// TIA Portal project "AP2_s71200" (V14)

(* hardware
DEVICE "S7-1200 station_1"  S7-1200 Station
   slot 0: "Rack_0"  S7-1200 Rack  Rack  V1.0
   slot 1: "PLC_1"  CPU 1214C DC/DC/DC  6ES7 214-1AG40-0XB0  V4.2
   slot 2: "DI 16/DQ 16x24VDC_1"  6ES7 223-1BL32-0XB0  V2.0
*)

// ===== PLC "PLC_1"  CPU 1214C DC/DC/DC =====

VAR_GLOBAL   // PLC tag table "Default tag table"
   "-F5" AT %I0.0 : Bool;
   "-S3" AT %I0.1 : Bool;
   "-S4" AT %I0.2 : Bool;
   "-S5" AT %I0.3 : Bool;
   "-S6" AT %I0.4 : Bool;
   "-S7" AT %I0.5 : Bool;
   "-S8" AT %I0.6 : Bool;
   "-S9" AT %I0.7 : Bool;
   "-S10" AT %I1.0 : Bool;
   "-S11" AT %I1.1 : Bool;
   "-S12" AT %I1.2 : Bool;
   "-BP1" AT %I1.3 : Bool;
   "-B11" AT %I1.4 : Bool;
   "-B12" AT %I1.5 : Bool;
   "-B13" AT %I2.0 : Bool;
   "-B21" AT %I2.1 : Bool;
   "-B22" AT %I2.2 : Bool;
   "-B31" AT %I2.3 : Bool;
   "-B32" AT %I2.4 : Bool;
   "Reserve1" AT %I2.5 : Bool;
   "Reserve2" AT %I2.6 : Bool;
   "Reserve3" AT %I2.7 : Bool;
   "Reserve4" AT %I3.0 : Bool;
   "-F7" AT %I3.1 : Bool;
   "-M21" AT %Q0.0 : Bool;
   "-M22" AT %Q0.1 : Bool;
   "-M31" AT %Q0.2 : Bool;
   "-M32" AT %Q0.3 : Bool;
   "Reserve5" AT %Q0.4 : Bool;
   "Reserve6" AT %Q0.5 : Bool;
   "-Q5" AT %Q0.6 : Bool;
   "-Q6" AT %Q0.7 : Bool;
   "-P32" AT %Q2.0 : Bool;
   "Reserve7" AT %Q2.1 : Bool;
   "-Q60" AT %Q2.2 : Bool;
   "-P2" AT %Q2.3 : Bool;
   "-P3" AT %Q2.4 : Bool;
   "-P4" AT %Q2.5 : Bool;
   "-P5" AT %Q2.6 : Bool;
   "-P6" AT %Q2.7 : Bool;
   "-P7" AT %Q3.0 : Bool;
   "-P8" AT %Q3.1 : Bool;
   "-P10" AT %Q3.2 : Bool;
   "-P11" AT %Q3.3 : Bool;
   "-P12" AT %Q3.4 : Bool;
   "-P13" AT %Q3.5 : Bool;
   "-P14" AT %Q3.6 : Bool;
   "-Reserve8" AT %Q3.7 : Bool;
   "G_Notification" AT %M0.0 : Bool;
   "G_Allow" AT %M0.1 : Bool;
   "Button" AT %M0.3 : Bool;
   "Auto" AT %M0.4 : Bool;
   "Allow" AT %M0.5 : Bool;
   "1Hz" AT %M0.6 : Bool;
   "T_Block" AT %M0.7 : Bool;
   "M21_A" AT %M1.0 : Bool;
   "M22_A" AT %M1.1 : Bool;
   "M31_A" AT %M1.2 : Bool;
   "M32_A" AT %M1.3 : Bool;
   "Q5_A" AT %M1.4 : Bool;
   "Q6_A" AT %M1.5 : Bool;
   "Q60_A" AT %M1.6 : Bool;
   "M21_B" AT %M1.7 : Bool;
   "M22_B" AT %M2.0 : Bool;
   "M31_B" AT %M2.1 : Bool;
   "M32_B" AT %M2.2 : Bool;
   "Q5_B" AT %M2.3 : Bool;
   "Q6_B" AT %M2.4 : Bool;
   "Q60_B" AT %M2.5 : Bool;
   "Out_Step 3" AT %M0.2 : Bool;
END_VAR

DATA_BLOCK "Clock_DB"   // DB3
{ S7_Optimized_Access := 'TRUE' }
VERSION : 0.1
// stored: InstanceOfName Clock
"Clock"
BEGIN
END_DATA_BLOCK

DATA_BLOCK "Safety_Activation_DB"   // DB4
{ S7_Optimized_Access := 'TRUE' }
VERSION : 0.1
// stored: InstanceOfName Safety_Activation
"Safety_Activation"
BEGIN
END_DATA_BLOCK

DATA_BLOCK "G_Allow__DB"   // DB5
{ S7_Optimized_Access := 'TRUE' }
VERSION : 0.1
// stored: InstanceOfName G_Allow_
"G_Allow_"
BEGIN
END_DATA_BLOCK

DATA_BLOCK "G_T_Block_DB"   // DB6
{ S7_Optimized_Access := 'TRUE' }
VERSION : 0.1
// stored: InstanceOfName G_T_Block
"G_T_Block"
BEGIN
END_DATA_BLOCK

DATA_BLOCK "G_Button_DB"   // DB7
{ S7_Optimized_Access := 'TRUE' }
VERSION : 0.1
// stored: InstanceOfName G_Button
"G_Button"
BEGIN
END_DATA_BLOCK

DATA_BLOCK "G_Notifications_DB"   // DB8
{ S7_Optimized_Access := 'TRUE' }
VERSION : 0.1
// stored: InstanceOfName G_Notifications
"G_Notifications"
BEGIN
END_DATA_BLOCK

DATA_BLOCK "G_Auto_DB"   // DB21
{ S7_Optimized_Access := 'TRUE' }
VERSION : 0.1
// stored: InstanceOfName G_Auto
"G_Auto"
BEGIN
END_DATA_BLOCK

DATA_BLOCK "Output_DB"   // DB22
{ S7_Optimized_Access := 'TRUE' }
VERSION : 0.1
// stored: InstanceOfName Output
"Output"
BEGIN
END_DATA_BLOCK

// folder: System blocks/Program resources

DATA_BLOCK "0.5s/X500"   // DB1
{ S7_Optimized_Access := 'TRUE' }
AUTHOR : Simatic
FAMILY : IEC
NAME : IEC_TMR
VERSION : 1.0
// stored: InstanceOfName IEC_TIMER
"IEC_TIMER"
BEGIN
END_DATA_BLOCK

DATA_BLOCK "0.5s/X501"   // DB2
{ S7_Optimized_Access := 'TRUE' }
AUTHOR : Simatic
FAMILY : IEC
NAME : IEC_TMR
VERSION : 1.0
// stored: InstanceOfName IEC_TIMER
"IEC_TIMER"
BEGIN
END_DATA_BLOCK

DATA_BLOCK "1s/B11_X301"   // DB9
{ S7_Optimized_Access := 'TRUE' }
AUTHOR : Simatic
FAMILY : IEC
NAME : IEC_TMR
VERSION : 1.0
// stored: InstanceOfName IEC_TIMER
"IEC_TIMER"
BEGIN
END_DATA_BLOCK

DATA_BLOCK "2s/B22_X302"   // DB10
{ S7_Optimized_Access := 'TRUE' }
AUTHOR : Simatic
FAMILY : IEC
NAME : IEC_TMR
VERSION : 1.0
// stored: InstanceOfName IEC_TIMER
"IEC_TIMER"
BEGIN
END_DATA_BLOCK

DATA_BLOCK "1s/B21_X303"   // DB11
{ S7_Optimized_Access := 'TRUE' }
AUTHOR : Simatic
FAMILY : IEC
NAME : IEC_TMR
VERSION : 1.0
// stored: InstanceOfName IEC_TIMER
"IEC_TIMER"
BEGIN
END_DATA_BLOCK

DATA_BLOCK "1s/B12_X304"   // DB12
{ S7_Optimized_Access := 'TRUE' }
AUTHOR : Simatic
FAMILY : IEC
NAME : IEC_TMR
VERSION : 1.0
// stored: InstanceOfName IEC_TIMER
"IEC_TIMER"
BEGIN
END_DATA_BLOCK

DATA_BLOCK "1s/B22_X305"   // DB13
{ S7_Optimized_Access := 'TRUE' }
AUTHOR : Simatic
FAMILY : IEC
NAME : IEC_TMR
VERSION : 1.0
// stored: InstanceOfName IEC_TIMER
"IEC_TIMER"
BEGIN
END_DATA_BLOCK

DATA_BLOCK "1s/B21_X308"   // DB14
{ S7_Optimized_Access := 'TRUE' }
AUTHOR : Simatic
FAMILY : IEC
NAME : IEC_TMR
VERSION : 1.0
// stored: InstanceOfName IEC_TIMER
"IEC_TIMER"
BEGIN
END_DATA_BLOCK

DATA_BLOCK "1s/B13_X309"   // DB15
{ S7_Optimized_Access := 'TRUE' }
AUTHOR : Simatic
FAMILY : IEC
NAME : IEC_TMR
VERSION : 1.0
// stored: InstanceOfName IEC_TIMER
"IEC_TIMER"
BEGIN
END_DATA_BLOCK

DATA_BLOCK "1s/B22_X310"   // DB16
{ S7_Optimized_Access := 'TRUE' }
AUTHOR : Simatic
FAMILY : IEC
NAME : IEC_TMR
VERSION : 1.0
// stored: InstanceOfName IEC_TIMER
"IEC_TIMER"
BEGIN
END_DATA_BLOCK

DATA_BLOCK "1s/X311"   // DB17
{ S7_Optimized_Access := 'TRUE' }
AUTHOR : Simatic
FAMILY : IEC
NAME : IEC_TMR
VERSION : 1.0
// stored: InstanceOfName IEC_TIMER
"IEC_TIMER"
BEGIN
END_DATA_BLOCK

DATA_BLOCK "1s/B21_X312"   // DB18
{ S7_Optimized_Access := 'TRUE' }
AUTHOR : Simatic
FAMILY : IEC
NAME : IEC_TMR
VERSION : 1.0
// stored: InstanceOfName IEC_TIMER
"IEC_TIMER"
BEGIN
END_DATA_BLOCK

DATA_BLOCK "2s/B31_X313"   // DB19
{ S7_Optimized_Access := 'TRUE' }
AUTHOR : Simatic
FAMILY : IEC
NAME : IEC_TMR
VERSION : 1.0
// stored: InstanceOfName IEC_TIMER
"IEC_TIMER"
BEGIN
END_DATA_BLOCK

DATA_BLOCK "1s/B32_X314"   // DB20
{ S7_Optimized_Access := 'TRUE' }
AUTHOR : Simatic
FAMILY : IEC
NAME : IEC_TMR
VERSION : 1.0
// stored: InstanceOfName IEC_TIMER
"IEC_TIMER"
BEGIN
END_DATA_BLOCK

// folder: (top level)

FUNCTION_BLOCK "Safety_Activation"   // FB1, FBD
{ S7_Optimized_Access := 'TRUE' }
VERSION : 0.1
   VAR_INPUT
      Allow : Bool;
      BP1 : Bool;
      S3 : Bool;
      S4 : Bool;
      F5 : Bool;
      F7 : Bool;
   END_VAR
   VAR_OUTPUT
      G_Notifications : Bool;
      G_Allow : Bool;
      "Out_step 3" : Bool;
      Button : Bool;
      Auto : Bool;
   END_VAR
   VAR
      "Step 1" : Bool;
      "Step 2" : Bool;
      "Step 3" : Bool;
      "Step 4" : Bool;
      "Step 5" : Bool;
   END_VAR
BEGIN

REGION Network 1
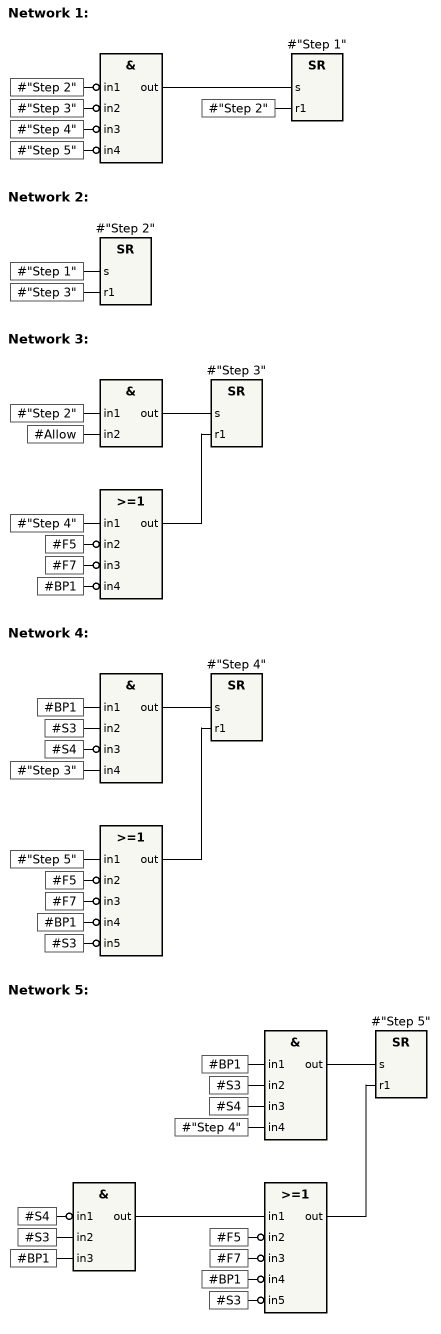
   IF NOT #"Step 2" AND NOT #"Step 3" AND NOT #"Step 4" AND NOT #"Step 5" THEN
       #"Step 1" := TRUE;   // SR flip-flop
   END_IF;
   IF #"Step 2" THEN #"Step 1" := FALSE; END_IF;
END_REGION

REGION Network 2
   IF #"Step 1" THEN
       #"Step 2" := TRUE;   // SR flip-flop
   END_IF;
   IF #"Step 3" THEN #"Step 2" := FALSE; END_IF;
END_REGION

REGION Network 3
   IF #"Step 2" AND #Allow THEN
       #"Step 3" := TRUE;   // SR flip-flop
   END_IF;
   IF #"Step 4" OR NOT #F5 OR NOT #F7 OR NOT #BP1 THEN #"Step 3" := FALSE; END_IF;
END_REGION

REGION Network 4
   IF #BP1 AND #S3 AND NOT #S4 AND #"Step 3" THEN
       #"Step 4" := TRUE;   // SR flip-flop
   END_IF;
   IF #"Step 5" OR NOT #F5 OR NOT #F7 OR NOT #BP1 OR NOT #S3 THEN #"Step 4" := FALSE; END_IF;
END_REGION

REGION Network 5
   IF #BP1 AND #S3 AND #S4 AND #"Step 4" THEN
       #"Step 5" := TRUE;   // SR flip-flop
   END_IF;
   IF (NOT #S4 AND #S3 AND #BP1) OR NOT #F5 OR NOT #F7 OR NOT #BP1 OR NOT #S3 THEN
       #"Step 5" := FALSE;
   END_IF;
END_REGION

REGION Network 6
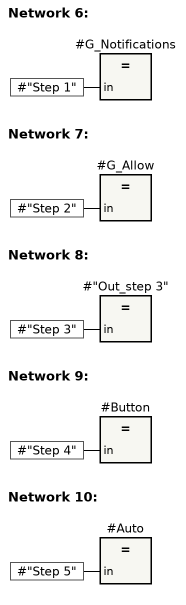
   #G_Notifications := #"Step 1";
END_REGION

REGION Network 7
   #G_Allow := #"Step 2";
END_REGION

REGION Network 8
   #"Out_step 3" := #"Step 3";
END_REGION

REGION Network 9
   #Button := #"Step 4";
END_REGION

REGION Network 10
   #Auto := #"Step 5";
END_REGION
END_FUNCTION_BLOCK

FUNCTION_BLOCK "Clock"   // FB2, FBD
{ S7_Optimized_Access := 'TRUE' }
VERSION : 0.1
   VAR_OUTPUT
      "1Hz" : Bool;
   END_VAR
   VAR
      "Step 500" : Bool;
      "Step 501" : Bool;
   END_VAR
BEGIN

REGION Network 1
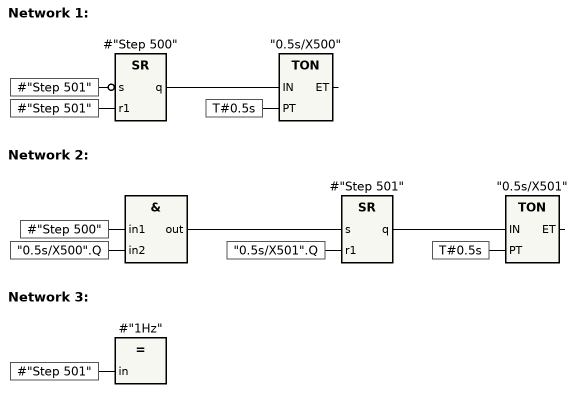
   IF NOT #"Step 501" THEN
       #"Step 500" := TRUE;   // SR flip-flop
   END_IF;
   IF #"Step 501" THEN #"Step 500" := FALSE; END_IF;
   "0.5s/X500".TON(IN := #"Step 500", PT := T#0.5s);
END_REGION

REGION Network 2
   IF #"Step 500" AND "0.5s/X500".Q THEN
       #"Step 501" := TRUE;   // SR flip-flop
   END_IF;
   IF "0.5s/X501".Q THEN #"Step 501" := FALSE; END_IF;
   "0.5s/X501".TON(IN := #"Step 501", PT := T#0.5s);
END_REGION

REGION Network 3
   #"1Hz" := #"Step 501";
END_REGION
END_FUNCTION_BLOCK

FUNCTION_BLOCK "G_Allow_"   // FB3, FBD
{ S7_Optimized_Access := 'TRUE' }
VERSION : 0.1
   VAR_INPUT
      G_Allow : Bool;
      "Out_step 3" : Bool;
      F5 : Bool;
      F7 : Bool;
      S4 : Bool;
      S5 : Bool;
      S6 : Bool;
      S7 : Bool;
      S8 : Bool;
      S9 : Bool;
      S10 : Bool;
      S12 : Bool;
   END_VAR
   VAR_OUTPUT
      Allow : Bool;
   END_VAR
   VAR
      "Step 50" : Bool;
      "Step 51" : Bool;
   END_VAR
BEGIN

REGION Network 1
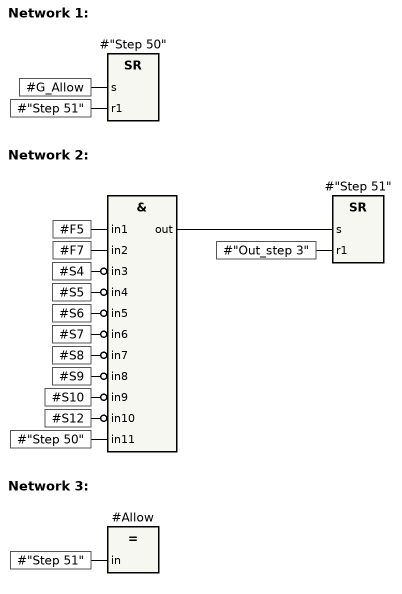
   IF #G_Allow THEN
       #"Step 50" := TRUE;   // SR flip-flop
   END_IF;
   IF #"Step 51" THEN #"Step 50" := FALSE; END_IF;
END_REGION

REGION Network 2
   IF #F5 AND #F7 AND NOT #S4 AND NOT #S5 AND NOT #S6 AND NOT #S7 AND NOT #S8 AND NOT #S9 AND NOT #S10 AND NOT #S12 AND #"Step 50" THEN
       #"Step 51" := TRUE;   // SR flip-flop
   END_IF;
   IF #"Out_step 3" THEN #"Step 51" := FALSE; END_IF;
END_REGION

REGION Network 3
   #Allow := #"Step 51";
END_REGION
END_FUNCTION_BLOCK

FUNCTION_BLOCK "G_T_Block"   // FB4, FBD
{ S7_Optimized_Access := 'TRUE' }
VERSION : 0.1
   VAR_INPUT
      Button : Bool;
      S6 : Bool;
      S7 : Bool;
   END_VAR
   VAR_OUTPUT
      T_Block : Bool;
   END_VAR
   VAR
      "Step 400" : Bool;
      "Step 401" : Bool;
   END_VAR
BEGIN

REGION Network 1
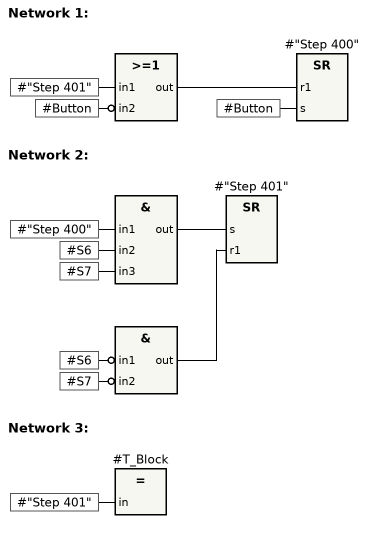
   IF #Button THEN
       #"Step 400" := TRUE;   // SR flip-flop
   END_IF;
   IF #"Step 401" OR NOT #Button THEN #"Step 400" := FALSE; END_IF;
END_REGION

REGION Network 2
   IF #"Step 400" AND #S6 AND #S7 THEN
       #"Step 401" := TRUE;   // SR flip-flop
   END_IF;
   IF NOT #S6 AND NOT #S7 THEN #"Step 401" := FALSE; END_IF;
END_REGION

REGION Network 3
   #T_Block := #"Step 401";
END_REGION
END_FUNCTION_BLOCK

FUNCTION_BLOCK "G_Button"   // FB5, FBD
{ S7_Optimized_Access := 'TRUE' }
VERSION : 0.1
   VAR_INPUT
      G_Button : Bool;
      G_T_Block : Bool;
      S6 : Bool;
      S7 : Bool;
      S8 : Bool;
      S9 : Bool;
      S10 : Bool;
      S12 : Bool;
      B11 : Bool;
      B13 : Bool;
      B21 : Bool;
      B22 : Bool;
      B31 : Bool;
      B32 : Bool;
      "Q5.in" : Bool;
      "Q6.in" : Bool;
   END_VAR
   VAR_OUTPUT
      Q5_B : Bool;
      Q6_B : Bool;
      M21_B : Bool;
      M22_B : Bool;
      M31_B : Bool;
      M32_B : Bool;
      Q60_B : Bool;
   END_VAR
   VAR
      "Step 200" : Bool;
   END_VAR
BEGIN

REGION Network 1
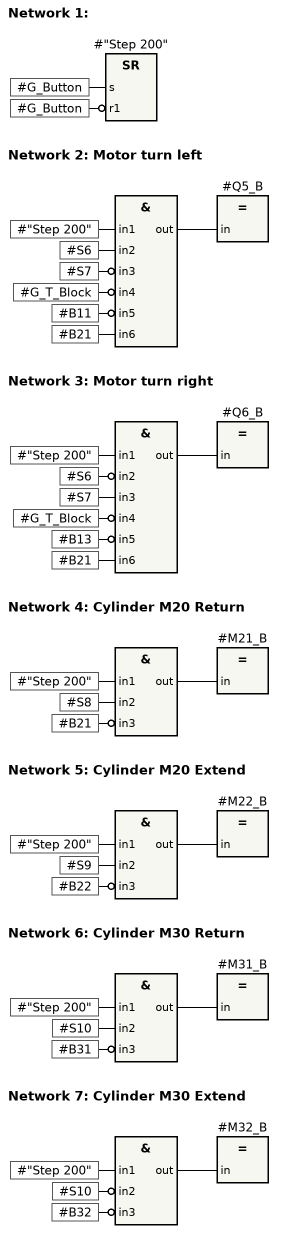
   IF #G_Button THEN
       #"Step 200" := TRUE;   // SR flip-flop
   END_IF;
   IF NOT #G_Button THEN #"Step 200" := FALSE; END_IF;
END_REGION

REGION Network 2: Motor turn left
   #Q5_B := #"Step 200" AND #S6 AND NOT #S7 AND NOT #G_T_Block AND NOT #B11 AND #B21;
END_REGION

REGION Network 3: Motor turn right
   #Q6_B := #"Step 200" AND NOT #S6 AND #S7 AND NOT #G_T_Block AND NOT #B13 AND #B21;
END_REGION

REGION Network 4: Cylinder M20 Return
   #M21_B := #"Step 200" AND #S8 AND NOT #B21;
END_REGION

REGION Network 5: Cylinder M20 Extend
   #M22_B := #"Step 200" AND #S9 AND NOT #B22;
END_REGION

REGION Network 6: Cylinder M30 Return
   #M31_B := #"Step 200" AND #S10 AND NOT #B31;
END_REGION

REGION Network 7: Cylinder M30 Extend
   #M32_B := #"Step 200" AND NOT #S10 AND NOT #B32;
END_REGION

REGION Network 8: Demagnetization
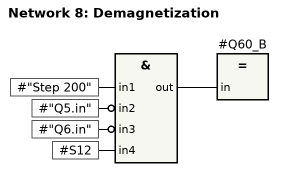
   #Q60_B := #"Step 200" AND NOT #"Q5.in" AND NOT #"Q6.in" AND #S12;
END_REGION
END_FUNCTION_BLOCK

FUNCTION_BLOCK "G_Notifications"   // FB6, FBD
{ S7_Optimized_Access := 'TRUE' }
VERSION : 0.1
   VAR_INPUT
      S3 : Bool;
      G_Notification : Bool;
      Auto : Bool;
      Button : Bool;
      "1Hz" : Bool;
      F7 : Bool;
      BP1 : Bool;
      B11 : Bool;
      B12 : Bool;
      B13 : Bool;
      B21 : Bool;
      B22 : Bool;
      B31 : Bool;
      B32 : Bool;
      "Q5.in" : Bool;
      "Q6.in" : Bool;
      "Q60.in" : Bool;
   END_VAR
   VAR_OUTPUT
      P2 : Bool;
      P3 : Bool;
      P4 : Bool;
      P5 : Bool;
      P6 : Bool;
      P7 : Bool;
      P8 : Bool;
      P10 : Bool;
      P11 : Bool;
      P12 : Bool;
      P13 : Bool;
      P14 : Bool;
      P32 : Bool;
   END_VAR
   VAR
      "Step 100" : Bool;
      "Step 101" : Bool;
   END_VAR
BEGIN

REGION Network 1
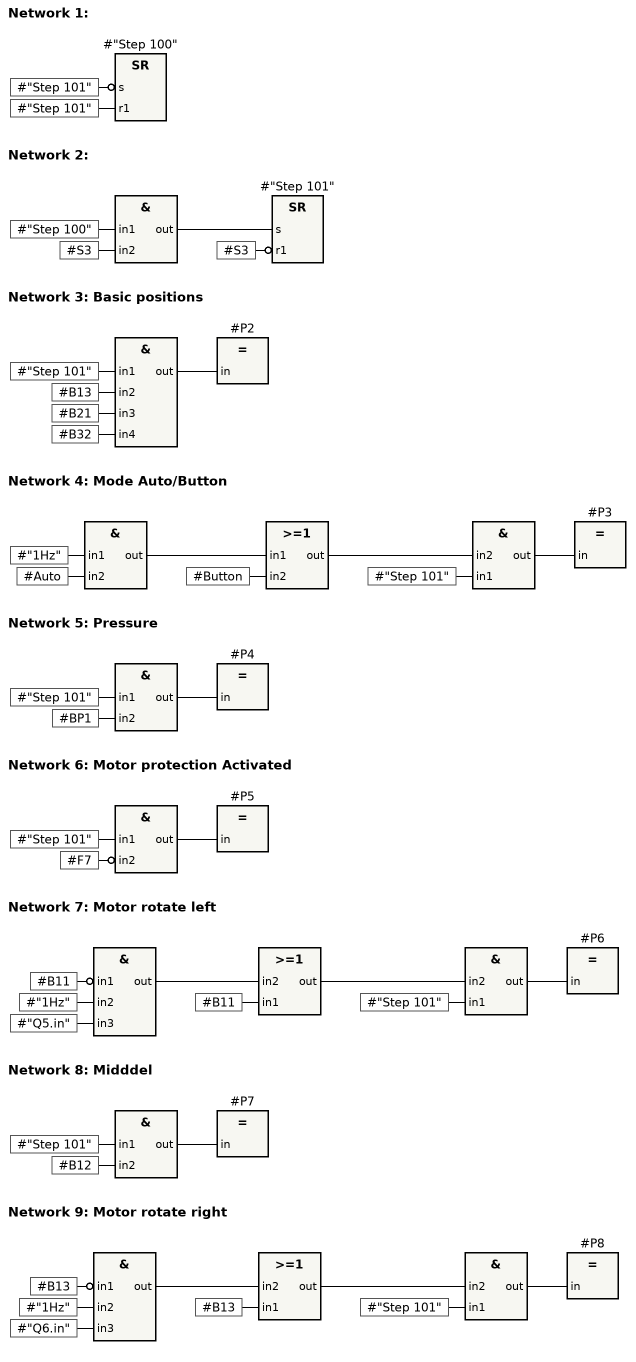
   IF NOT #"Step 101" THEN
       #"Step 100" := TRUE;   // SR flip-flop
   END_IF;
   IF #"Step 101" THEN #"Step 100" := FALSE; END_IF;
END_REGION

REGION Network 2
   IF #"Step 100" AND #S3 THEN
       #"Step 101" := TRUE;   // SR flip-flop
   END_IF;
   IF NOT #S3 THEN #"Step 101" := FALSE; END_IF;
END_REGION

REGION Network 3: Basic positions
   #P2 := #"Step 101" AND #B13 AND #B21 AND #B32;
END_REGION

REGION Network 4: Mode Auto/Button
   #P3 := ((#"1Hz" AND #Auto) OR #Button) AND #"Step 101";
END_REGION

REGION Network 5: Pressure
   #P4 := #"Step 101" AND #BP1;
END_REGION

REGION Network 6: Motor protection Activated
   #P5 := #"Step 101" AND NOT #F7;
END_REGION

REGION Network 7: Motor rotate left
   #P6 := ((NOT #B11 AND #"1Hz" AND #"Q5.in") OR #B11) AND #"Step 101";
END_REGION

REGION Network 8: Midddel
   #P7 := #"Step 101" AND #B12;
END_REGION

REGION Network 9: Motor rotate right
   #P8 := ((NOT #B13 AND #"1Hz" AND #"Q6.in") OR #B13) AND #"Step 101";
END_REGION

REGION Network 10: M20 In
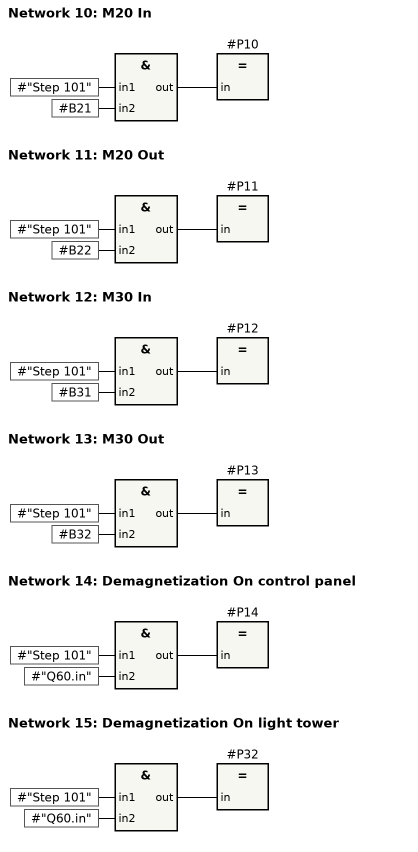
   #P10 := #"Step 101" AND #B21;
END_REGION

REGION Network 11: M20 Out
   #P11 := #"Step 101" AND #B22;
END_REGION

REGION Network 12: M30 In
   #P12 := #"Step 101" AND #B31;
END_REGION

REGION Network 13: M30 Out
   // ADD In
   #P13 := #"Step 101" AND #B32;
END_REGION

REGION Network 14: Demagnetization On control panel
   #P14 := #"Step 101" AND #"Q60.in";
END_REGION

REGION Network 15: Demagnetization On light tower
   #P32 := #"Step 101" AND #"Q60.in";
END_REGION
END_FUNCTION_BLOCK

FUNCTION_BLOCK "G_Auto"   // FB7, FBD
{ S7_Optimized_Access := 'TRUE' }
VERSION : 0.1
   VAR_INPUT
      Auto : Bool;
      S5 : Bool;
      B11 : Bool;
      B12 : Bool;
      B13 : Bool;
      B21 : Bool;
      B22 : Bool;
      B31 : Bool;
      B32 : Bool;
   END_VAR
   VAR_OUTPUT
      M21_A : Bool;
      M22_A : Bool;
      M31_A : Bool;
      M32_A : Bool;
      Q5_A : Bool;
      Q6_A : Bool;
      Q60_A : Bool;
   END_VAR
   VAR
      "Step 300" : Bool;
      "Step 301" : Bool;
      "Step 302" : Bool;
      "Step 303" : Bool;
      "Step 304" : Bool;
      "Step 305" : Bool;
      "Step 306" : Bool;
      "Step 307" : Bool;
      "Step 308" : Bool;
      "Step 309" : Bool;
      "Step 310" : Bool;
      "Step 311" : Bool;
      "Step 312" : Bool;
      "Step 313" : Bool;
      "Step 314" : Bool;
   END_VAR
BEGIN

REGION Network 1
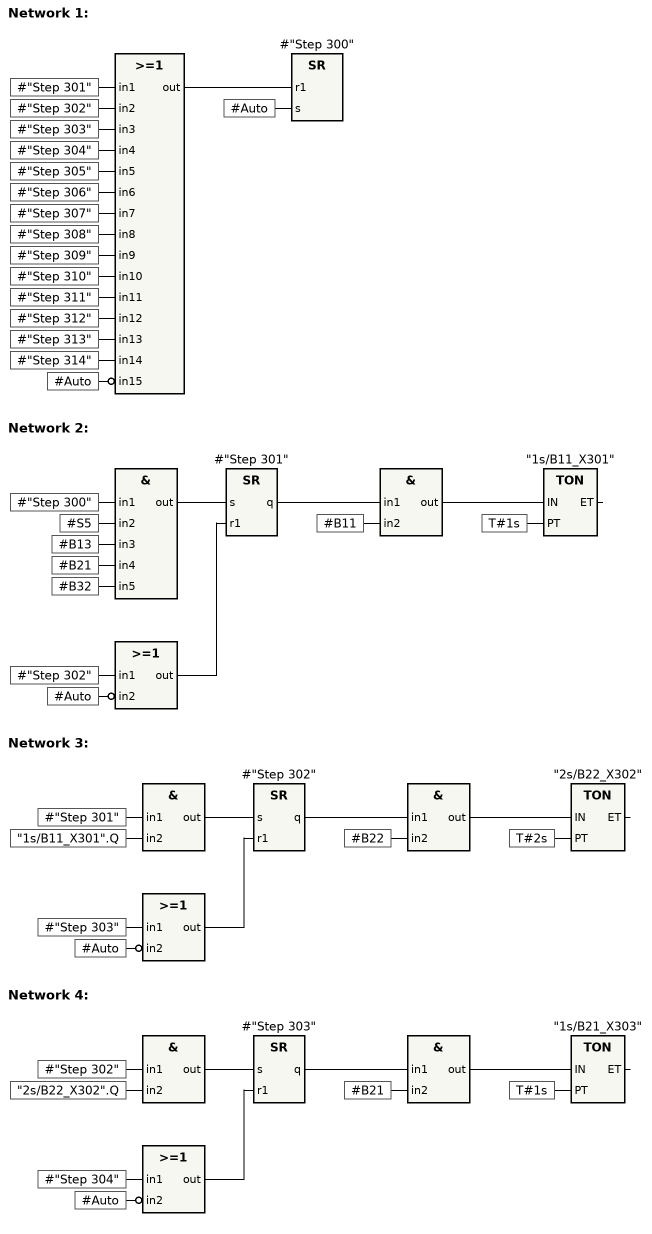
   IF #Auto THEN
       #"Step 300" := TRUE;   // SR flip-flop
   END_IF;
   IF #"Step 301" OR #"Step 302" OR #"Step 303" OR #"Step 304" OR #"Step 305" OR #"Step 306" OR #"Step 307" OR #"Step 308" OR #"Step 309" OR #"Step 310" OR #"Step 311" OR #"Step 312" OR #"Step 313" OR #"Step 314" OR NOT #Auto THEN
       #"Step 300" := FALSE;
   END_IF;
END_REGION

REGION Network 2
   IF #"Step 300" AND #S5 AND #B13 AND #B21 AND #B32 THEN
       #"Step 301" := TRUE;   // SR flip-flop
   END_IF;
   IF #"Step 302" OR NOT #Auto THEN #"Step 301" := FALSE; END_IF;
   "1s/B11_X301".TON(IN := #"Step 301" AND #B11, PT := T#1s);
END_REGION

REGION Network 3
   IF #"Step 301" AND "1s/B11_X301".Q THEN
       #"Step 302" := TRUE;   // SR flip-flop
   END_IF;
   IF #"Step 303" OR NOT #Auto THEN #"Step 302" := FALSE; END_IF;
   "2s/B22_X302".TON(IN := #"Step 302" AND #B22, PT := T#2s);
END_REGION

REGION Network 4
   IF #"Step 302" AND "2s/B22_X302".Q THEN
       #"Step 303" := TRUE;   // SR flip-flop
   END_IF;
   IF #"Step 304" OR NOT #Auto THEN #"Step 303" := FALSE; END_IF;
   "1s/B21_X303".TON(IN := #"Step 303" AND #B21, PT := T#1s);
END_REGION

REGION Network 5
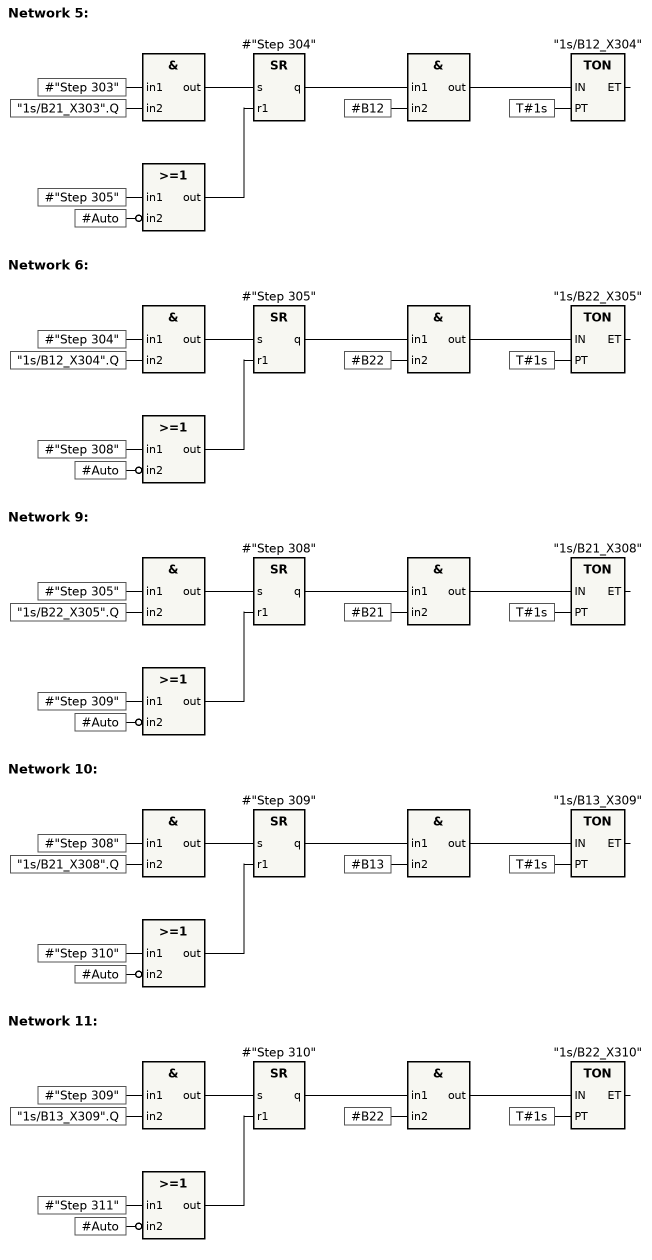
   IF #"Step 303" AND "1s/B21_X303".Q THEN
       #"Step 304" := TRUE;   // SR flip-flop
   END_IF;
   IF #"Step 305" OR NOT #Auto THEN #"Step 304" := FALSE; END_IF;
   "1s/B12_X304".TON(IN := #"Step 304" AND #B12, PT := T#1s);
END_REGION

REGION Network 6
   IF #"Step 304" AND "1s/B12_X304".Q THEN
       #"Step 305" := TRUE;   // SR flip-flop
   END_IF;
   IF #"Step 308" OR NOT #Auto THEN #"Step 305" := FALSE; END_IF;
   "1s/B22_X305".TON(IN := #"Step 305" AND #B22, PT := T#1s);
END_REGION

REGION Network 9
   IF #"Step 305" AND "1s/B22_X305".Q THEN
       #"Step 308" := TRUE;   // SR flip-flop
   END_IF;
   IF #"Step 309" OR NOT #Auto THEN #"Step 308" := FALSE; END_IF;
   "1s/B21_X308".TON(IN := #"Step 308" AND #B21, PT := T#1s);
END_REGION

REGION Network 10
   IF #"Step 308" AND "1s/B21_X308".Q THEN
       #"Step 309" := TRUE;   // SR flip-flop
   END_IF;
   IF #"Step 310" OR NOT #Auto THEN #"Step 309" := FALSE; END_IF;
   "1s/B13_X309".TON(IN := #"Step 309" AND #B13, PT := T#1s);
END_REGION

REGION Network 11
   IF #"Step 309" AND "1s/B13_X309".Q THEN
       #"Step 310" := TRUE;   // SR flip-flop
   END_IF;
   IF #"Step 311" OR NOT #Auto THEN #"Step 310" := FALSE; END_IF;
   "1s/B22_X310".TON(IN := #"Step 310" AND #B22, PT := T#1s);
END_REGION

REGION Network 12
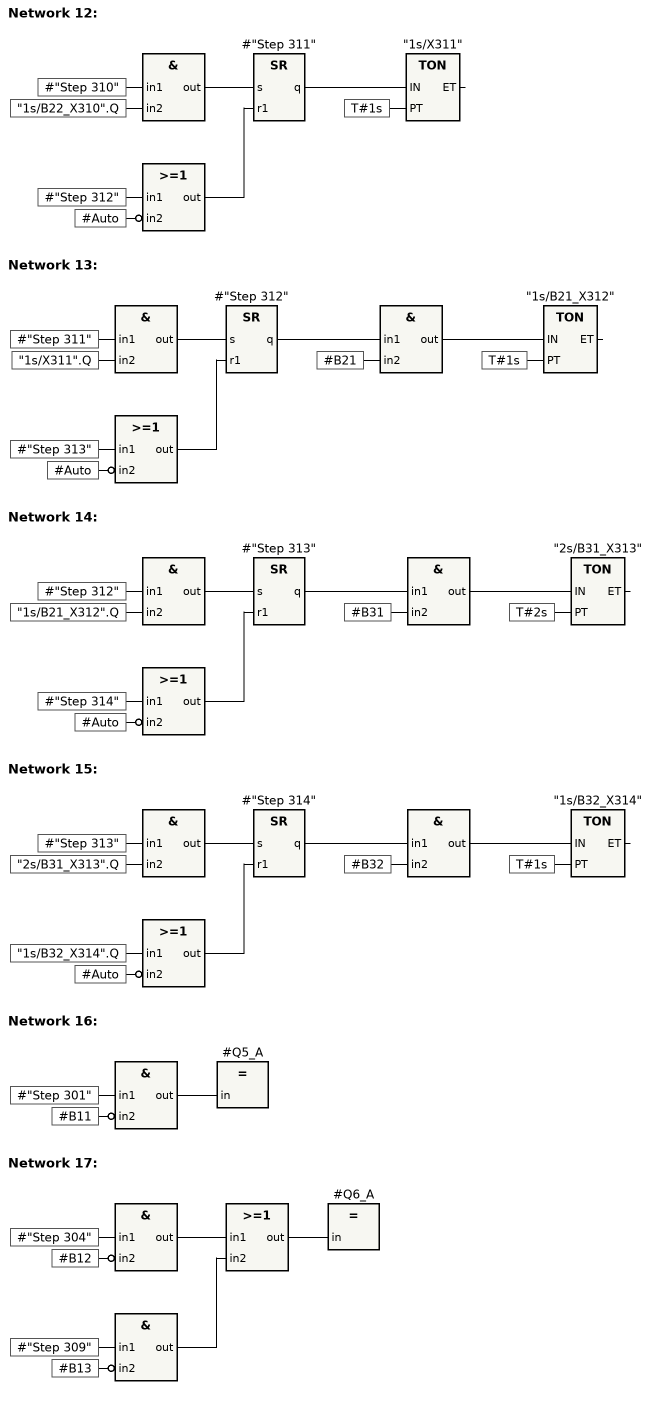
   IF #"Step 310" AND "1s/B22_X310".Q THEN
       #"Step 311" := TRUE;   // SR flip-flop
   END_IF;
   IF #"Step 312" OR NOT #Auto THEN #"Step 311" := FALSE; END_IF;
   "1s/X311".TON(IN := #"Step 311", PT := T#1s);
END_REGION

REGION Network 13
   IF #"Step 311" AND "1s/X311".Q THEN
       #"Step 312" := TRUE;   // SR flip-flop
   END_IF;
   IF #"Step 313" OR NOT #Auto THEN #"Step 312" := FALSE; END_IF;
   "1s/B21_X312".TON(IN := #"Step 312" AND #B21, PT := T#1s);
END_REGION

REGION Network 14
   IF #"Step 312" AND "1s/B21_X312".Q THEN
       #"Step 313" := TRUE;   // SR flip-flop
   END_IF;
   IF #"Step 314" OR NOT #Auto THEN #"Step 313" := FALSE; END_IF;
   "2s/B31_X313".TON(IN := #"Step 313" AND #B31, PT := T#2s);
END_REGION

REGION Network 15
   IF #"Step 313" AND "2s/B31_X313".Q THEN
       #"Step 314" := TRUE;   // SR flip-flop
   END_IF;
   IF "1s/B32_X314".Q OR NOT #Auto THEN #"Step 314" := FALSE; END_IF;
   "1s/B32_X314".TON(IN := #"Step 314" AND #B32, PT := T#1s);
END_REGION

REGION Network 16
   #Q5_A := #"Step 301" AND NOT #B11;
END_REGION

REGION Network 17
   #Q6_A := (#"Step 304" AND NOT #B12) OR (#"Step 309" AND NOT #B13);
END_REGION

REGION Network 18
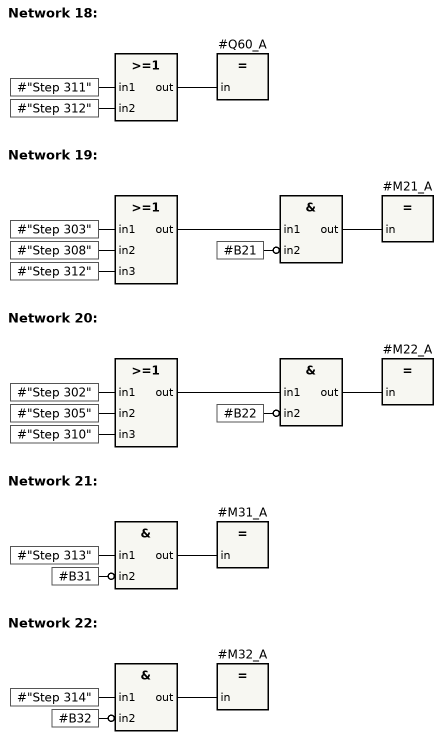
   #Q60_A := #"Step 311" OR #"Step 312";
END_REGION

REGION Network 19
   #M21_A := (#"Step 303" OR #"Step 308" OR #"Step 312") AND NOT #B21;
END_REGION

REGION Network 20
   #M22_A := (#"Step 302" OR #"Step 305" OR #"Step 310") AND NOT #B22;
END_REGION

REGION Network 21
   #M31_A := #"Step 313" AND NOT #B31;
END_REGION

REGION Network 22
   #M32_A := #"Step 314" AND NOT #B32;
END_REGION
END_FUNCTION_BLOCK

FUNCTION_BLOCK "Output"   // FB8, FBD
{ S7_Optimized_Access := 'TRUE' }
VERSION : 0.1
   VAR_INPUT
      M21_A : Bool;
      M22_A : Bool;
      M31_A : Bool;
      M32_A : Bool;
      Q5_A : Bool;
      Q6_A : Bool;
      Q60_A : Bool;
      Q5_B : Bool;
      Q6_B : Bool;
      M21_B : Bool;
      M22_B : Bool;
      M31_B : Bool;
      M32_B : Bool;
      Q60_B : Bool;
   END_VAR
   VAR_OUTPUT
      M21 : Bool;
      M22 : Bool;
      M31 : Bool;
      M32 : Bool;
      Q5 : Bool;
      Q6 : Bool;
      Q60 : Bool;
   END_VAR
BEGIN

REGION Network 1
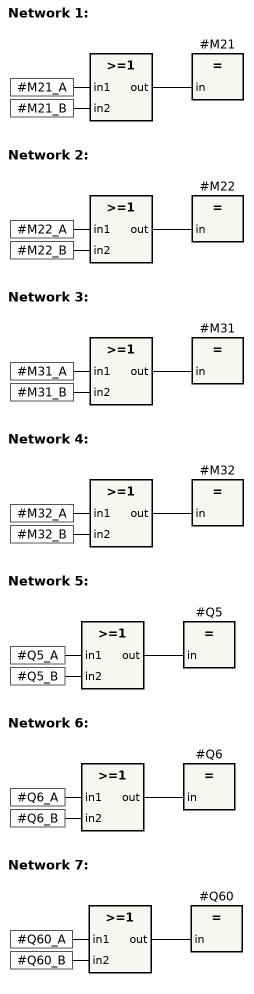
   #M21 := #M21_A OR #M21_B;
END_REGION

REGION Network 2
   #M22 := #M22_A OR #M22_B;
END_REGION

REGION Network 3
   #M31 := #M31_A OR #M31_B;
END_REGION

REGION Network 4
   #M32 := #M32_A OR #M32_B;
END_REGION

REGION Network 5
   #Q5 := #Q5_A OR #Q5_B;
END_REGION

REGION Network 6
   #Q6 := #Q6_A OR #Q6_B;
END_REGION

REGION Network 7
   #Q60 := #Q60_A OR #Q60_B;
END_REGION
END_FUNCTION_BLOCK

ORGANIZATION_BLOCK "Main"   // OB1, FBD, ProgramCycle
TITLE = "Main Program Sweep (Cycle)"
{ S7_Optimized_Access := 'TRUE' }
VERSION : 0.1
   VAR_INPUT
      Initial_Call : Bool;   // Initial call of this OB
      Remanence : Bool;   // =True, if remanent data are available
   END_VAR
BEGIN

REGION Network 1: Pluse
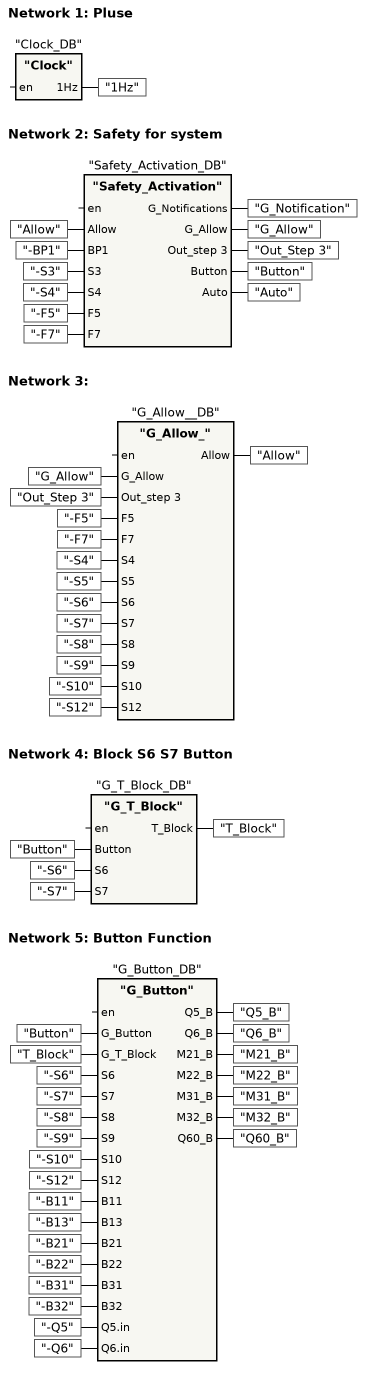
   "Clock_DB"("1Hz" => "1Hz");   // "Clock"
END_REGION

REGION Network 2: Safety for system
   "Safety_Activation_DB"(Allow := "Allow",   // "Safety_Activation"
                          BP1 := "-BP1",
                          S3 := "-S3",
                          S4 := "-S4",
                          F5 := "-F5",
                          F7 := "-F7",
                          G_Notifications => "G_Notification",
                          G_Allow => "G_Allow",
                          "Out_step 3" => "Out_Step 3",
                          Button => "Button",
                          Auto => "Auto");
END_REGION

REGION Network 3
   "G_Allow__DB"(G_Allow := "G_Allow",   // "G_Allow_"
                 "Out_step 3" := "Out_Step 3",
                 F5 := "-F5",
                 F7 := "-F7",
                 S4 := "-S4",
                 S5 := "-S5",
                 S6 := "-S6",
                 S7 := "-S7",
                 S8 := "-S8",
                 S9 := "-S9",
                 S10 := "-S10",
                 S12 := "-S12",
                 Allow => "Allow");
END_REGION

REGION Network 4: Block S6 S7 Button
   "G_T_Block_DB"(Button := "Button", S6 := "-S6", S7 := "-S7", T_Block => "T_Block");   // "G_T_Block"
END_REGION

REGION Network 5: Button Function
   "G_Button_DB"(G_Button := "Button",   // "G_Button"
                 G_T_Block := "T_Block",
                 S6 := "-S6",
                 S7 := "-S7",
                 S8 := "-S8",
                 S9 := "-S9",
                 S10 := "-S10",
                 S12 := "-S12",
                 B11 := "-B11",
                 B13 := "-B13",
                 B21 := "-B21",
                 B22 := "-B22",
                 B31 := "-B31",
                 B32 := "-B32",
                 "Q5.in" := "-Q5",
                 "Q6.in" := "-Q6",
                 Q5_B => "Q5_B",
                 Q6_B => "Q6_B",
                 M21_B => "M21_B",
                 M22_B => "M22_B",
                 M31_B => "M31_B",
                 M32_B => "M32_B",
                 Q60_B => "Q60_B");
END_REGION

REGION Network 6: Indicator
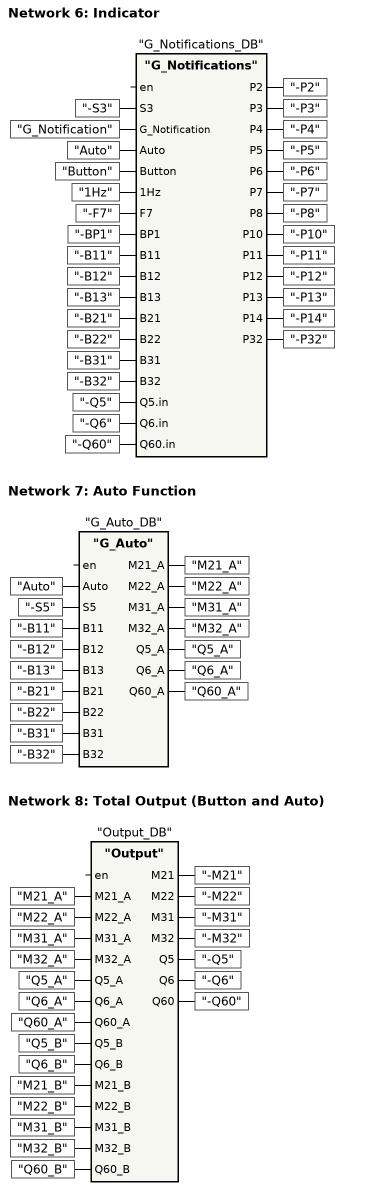
   "G_Notifications_DB"(S3 := "-S3",   // "G_Notifications"
                        G_Notification := "G_Notification",
                        Auto := "Auto",
                        Button := "Button",
                        "1Hz" := "1Hz",
                        F7 := "-F7",
                        BP1 := "-BP1",
                        B11 := "-B11",
                        B12 := "-B12",
                        B13 := "-B13",
                        B21 := "-B21",
                        B22 := "-B22",
                        B31 := "-B31",
                        B32 := "-B32",
                        "Q5.in" := "-Q5",
                        "Q6.in" := "-Q6",
                        "Q60.in" := "-Q60",
                        P2 => "-P2",
                        P3 => "-P3",
                        P4 => "-P4",
                        P5 => "-P5",
                        P6 => "-P6",
                        P7 => "-P7",
                        P8 => "-P8",
                        P10 => "-P10",
                        P11 => "-P11",
                        P12 => "-P12",
                        P13 => "-P13",
                        P14 => "-P14",
                        P32 => "-P32");
END_REGION

REGION Network 7: Auto Function
   "G_Auto_DB"(Auto := "Auto",   // "G_Auto"
               S5 := "-S5",
               B11 := "-B11",
               B12 := "-B12",
               B13 := "-B13",
               B21 := "-B21",
               B22 := "-B22",
               B31 := "-B31",
               B32 := "-B32",
               M21_A => "M21_A",
               M22_A => "M22_A",
               M31_A => "M31_A",
               M32_A => "M32_A",
               Q5_A => "Q5_A",
               Q6_A => "Q6_A",
               Q60_A => "Q60_A");
END_REGION

REGION Network 8: Total Output (Button and Auto)
   "Output_DB"(M21_A := "M21_A",   // "Output"
               M22_A := "M22_A",
               M31_A := "M31_A",
               M32_A := "M32_A",
               Q5_A := "Q5_A",
               Q6_A := "Q6_A",
               Q60_A := "Q60_A",
               Q5_B := "Q5_B",
               Q6_B := "Q6_B",
               M21_B := "M21_B",
               M22_B := "M22_B",
               M31_B := "M31_B",
               M32_B := "M32_B",
               Q60_B := "Q60_B",
               M21 => "-M21",
               M22 => "-M22",
               M31 => "-M31",
               M32 => "-M32",
               Q5 => "-Q5",
               Q6 => "-Q6",
               Q60 => "-Q60");
END_REGION
END_ORGANIZATION_BLOCK